VISUALIZATION Motor  // 2x2
END_VISUALIZATION

(* stored: Version 1.1.0.1, ProductVersion 3.1.0.26
   Visu Motor: Id {2d239a21-6786-4300-a739-aeccadb5952a} *)
